// TIA Portal V19 export
TYPE "TMeasuring_STATUSWORD"
// stored: Access Published
   STRUCT
      Control : Bool;   // 0: Technology object not in operation; 1: Technology object in operation
      Error : Bool;   // 0: No "Restart" active; 1: Change to "Restart" tags. For the changes to be applied, the technology
      RestartActive : Bool;   // 0: No "Restart" active; 1: Change to "Restart" tags. For the changes to be applied, the technology
      OnlineStartValuesChanged : Bool;   // Data record written with SFB WRREC
      CommunicationOK : Bool;   // Commando "Write"
   END_STRUCT;
END_TYPE
